// TIA Portal V20 export
TYPE "typeSequenceControlNodetransferPnPRightJobInterface_GRnR"
// stored: Namespace Unit1.Em5
   STRUCT
      hipotThicknessPICKJob5 : "LER_typeJobInterface";
      visionPLACEJob6 : "LER_typeJobInterface";
      visionPICKJob7 : "LER_typeJobInterface";
      weightCheckPLACEJob8 : "LER_typeJobInterface";
      weightCheckPICKJob9 : "LER_typeJobInterface";
   END_STRUCT;
END_TYPE
